// TIA Portal V18 export
FUNCTION "AHUDemands" : Void   // FC60008, LAD
{ S7_Optimized_Access := 'TRUE' }
VERSION : 0.1
// stored: AutoNumber false, IsIECCheckEnabled false, SetENOAutomatically false, UDAEnableTagReadback false
   VAR_INPUT
      iUnitID : Int;
      cHeatingRegState : Byte;
      cCoolingRegState : Byte;
      cIAQRegState : Byte;
      cBuildingdPRegState : Byte;
   END_VAR
   VAR_OUTPUT
      rHeaterDemand : Real;
      rCoolerDemand : Real;
      rFreshAirDemand : Real;
   END_VAR
BEGIN

REGION Network 1: Temperature demands(0-100%) defining (PID)
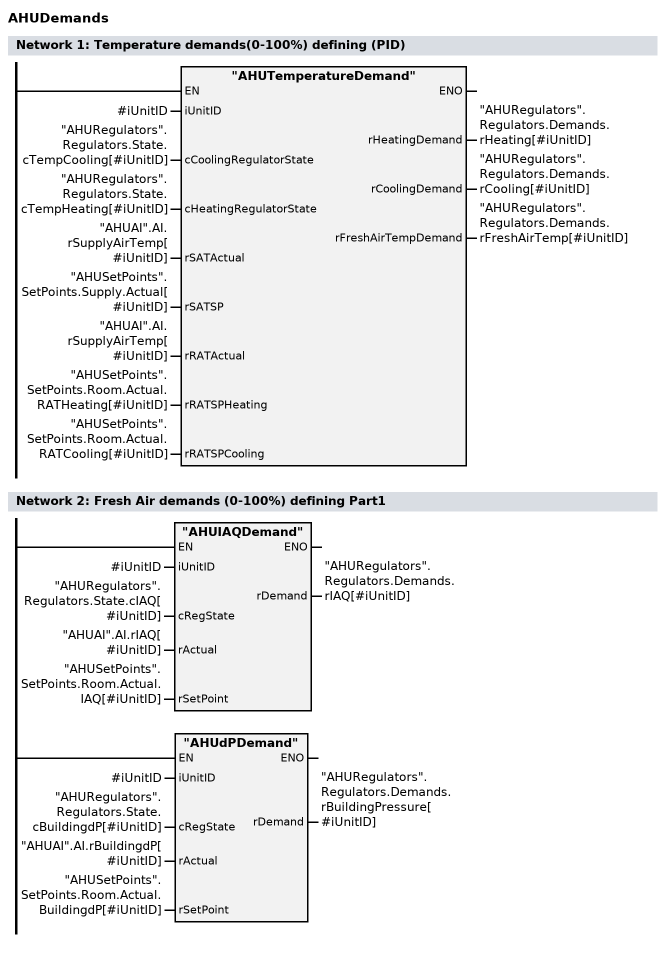
   RUNG wire#powerrail
      "AHUTemperatureDemand"(iUnitID := #iUnitID, cCoolingRegulatorState := "AHURegulators".Regulators.State.cTempCooling[#iUnitID], cHeatingRegulatorState := "AHURegulators".Regulators.State.cTempHeating[#iUnitID], rSATActual := "AHUAI".AI.rSupplyAirTemp[#iUnitID], rSATSP := "AHUSetPoints".SetPoints.Supply.Actual[#iUnitID], rRATActual := "AHUAI".AI.rSupplyAirTemp[#iUnitID], rRATSPHeating := "AHUSetPoints".SetPoints.Room.Actual.RATHeating[#iUnitID], rRATSPCooling := "AHUSetPoints".SetPoints.Room.Actual.RATCooling[#iUnitID], rHeatingDemand => "AHURegulators".Regulators.Demands.rHeating[#iUnitID], rCoolingDemand => "AHURegulators".Regulators.Demands.rCooling[#iUnitID], rFreshAirTempDemand => "AHURegulators".Regulators.Demands.rFreshAirTemp[#iUnitID])
   END_RUNG
   // the same network as SCL:
   "AHUTemperatureDemand"(iUnitID := #iUnitID,
                          cCoolingRegulatorState := "AHURegulators".Regulators.State.cTempCooling[#iUnitID],
                          cHeatingRegulatorState := "AHURegulators".Regulators.State.cTempHeating[#iUnitID],
                          rSATActual := "AHUAI".AI.rSupplyAirTemp[#iUnitID],
                          rSATSP := "AHUSetPoints".SetPoints.Supply.Actual[#iUnitID],
                          rRATActual := "AHUAI".AI.rSupplyAirTemp[#iUnitID],
                          rRATSPHeating := "AHUSetPoints".SetPoints.Room.Actual.RATHeating[#iUnitID],
                          rRATSPCooling := "AHUSetPoints".SetPoints.Room.Actual.RATCooling[#iUnitID],
                          rHeatingDemand => "AHURegulators".Regulators.Demands.rHeating[#iUnitID],
                          rCoolingDemand => "AHURegulators".Regulators.Demands.rCooling[#iUnitID],
                          rFreshAirTempDemand => "AHURegulators".Regulators.Demands.rFreshAirTemp[#iUnitID]);
END_REGION

REGION Network 2: Fresh Air demands (0-100%) defining Part1
   RUNG wire#powerrail
      "AHUIAQDemand"(iUnitID := #iUnitID, cRegState := "AHURegulators".Regulators.State.cIAQ[#iUnitID], rActual := "AHUAI".AI.rIAQ[#iUnitID], rSetPoint := "AHUSetPoints".SetPoints.Room.Actual.IAQ[#iUnitID], rDemand => "AHURegulators".Regulators.Demands.rIAQ[#iUnitID])
   END_RUNG
   RUNG wire#powerrail
      "AHUdPDemand"(iUnitID := #iUnitID, cRegState := "AHURegulators".Regulators.State.cBuildingdP[#iUnitID], rActual := "AHUAI".AI.rBuildingdP[#iUnitID], rSetPoint := "AHUSetPoints".SetPoints.Room.Actual.BuildingdP[#iUnitID], rDemand => "AHURegulators".Regulators.Demands.rBuildingPressure[#iUnitID])
   END_RUNG
   // the same network as SCL:
   "AHUIAQDemand"(iUnitID := #iUnitID,
                  cRegState := "AHURegulators".Regulators.State.cIAQ[#iUnitID],
                  rActual := "AHUAI".AI.rIAQ[#iUnitID],
                  rSetPoint := "AHUSetPoints".SetPoints.Room.Actual.IAQ[#iUnitID],
                  rDemand => "AHURegulators".Regulators.Demands.rIAQ[#iUnitID]);
   "AHUdPDemand"(iUnitID := #iUnitID,
                 cRegState := "AHURegulators".Regulators.State.cBuildingdP[#iUnitID],
                 rActual := "AHUAI".AI.rBuildingdP[#iUnitID],
                 rSetPoint := "AHUSetPoints".SetPoints.Room.Actual.BuildingdP[#iUnitID],
                 rDemand => "AHURegulators".Regulators.Demands.rBuildingPressure[#iUnitID]);
END_REGION

REGION Network 3 (SCL): Fresh Air demands defining Part2
   (* "AHUDmnds".Demands.rFreshAir[#iUnitID] := MAX(IN1 := "AHUDmnds".Demands.rIAQ[#iUnitID] * "AHUFreshAirCoef".FreshAirCoef.IAQ[#iUnitID],
                                                IN2 := "AHUDmnds".Demands.rBuildingPressure[#iUnitID] * "AHUFreshAirCoef".FreshAirCoef.BuildingdP[#iUnitID],
                                                IN3 := "AHUDmnds".Demands.rFreshAirTemp[#iUnitID] * "AHUFreshAirCoef".FreshAirCoef.Temperature[#iUnitID]); *)
END_REGION
END_FUNCTION
